FUNCTION_BLOCK AssemblySequenceAutomatic EXTENDS AssemblySequence IMPLEMENTS ZCore.ISequence
VAR
  _step : ZCore.Step(AssemblyStep.AutomaticBegin, AssemblyStep.AutomaticEnd);
END_VAR

IF NOT Busy THEN
  RETURN;
END_IF

IF OnStart(_step) THEN
  ; // init custom sequence variables here ...
END_IF

IF OnStop() THEN
  RETURN; // external stop was triggered
END_IF

IF OnHalt() THEN
  ; // Halting := TRUE; // Uncomment to acknowledge that the sequence is halting
END_IF

REPEAT
  LogStep();

  CASE _step.Index OF
    (* -------------------------------------------------------------------------------------------------------------------------------- *)
    AssemblyStep.AutomaticBegin:
    (* -------------------------------------------------------------------------------------------------------------------------------- *)
      IF _step.OnEntry()
      THEN
        ;
      END_IF

      // Await(obj1:=, nextStep:=AssemblyStep.AutomaticEnd);
      _step.SetNext(AssemblyStep.AutomaticEnd);
    
    (* -------------------------------------------------------------------------------------------------------------------------------- *)
    AssemblyStep.AutomaticEnd:
    (* -------------------------------------------------------------------------------------------------------------------------------- *)
      SetBusy(FALSE);
  
  ELSE
    Abort('sequence contains unhandled step');
  END_CASE
UNTIL _step.IsNotRepeatable() OR_ELSE NOT Busy END_REPEAT

END_FUNCTION_BLOCK

(* stored: Version 1.1.0.1
   POU AssemblySequenceAutomatic: Id {b0601c37-d6d9-41d7-a487-c2e3aca00399}, SpecialFunc None *)
